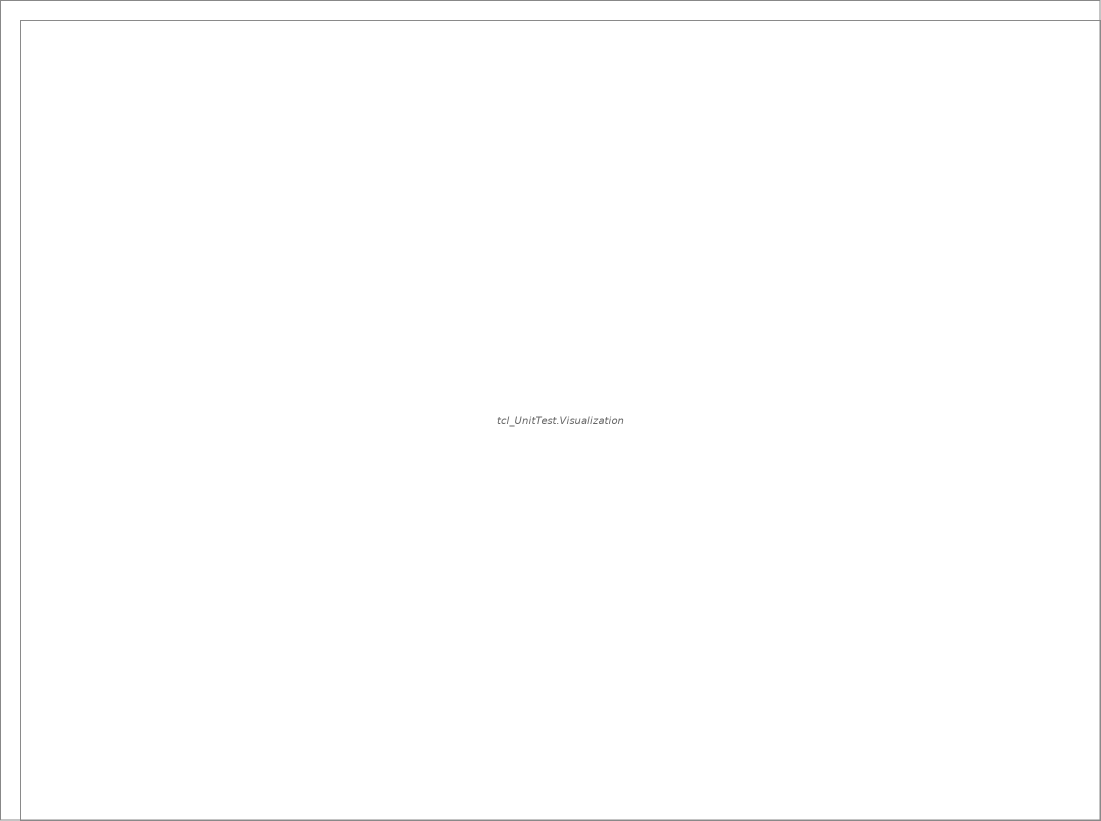
VISUALIZATION Visualization  // 1101x821
    Frame (20,20 1081x801)
        shows tcl_UnitTest.Visualization()
END_VISUALIZATION

(* stored: Version 1.1.0.1, ProductVersion 3.1.4024.3
   Visu Visualization: Id {62c33ba5-c696-471a-8e4f-5bc08ac8d7ba} *)
